// LS Electric XG5000 project: 과년67_2_4
// PLC NewPLC
// module base 0 slot 0: 입출력 모듈:XBC-DR20S (DC 24V 입력 12점, 릴레이 출력 8점)

PROGRAM NewProgram (task: 스캔 프로그램)

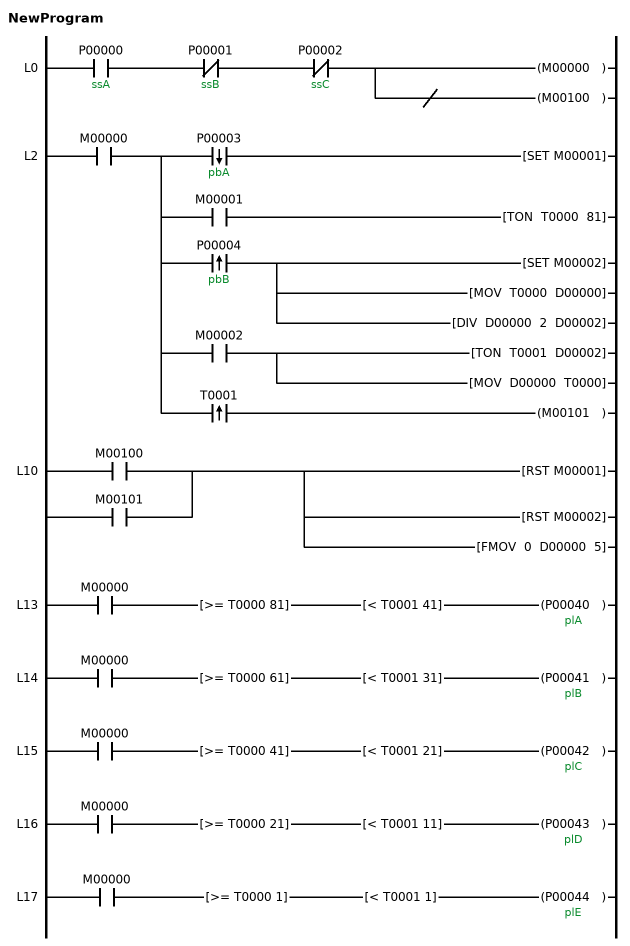
; L0
LOAD      P00000	// ssA
AND NOT   P00001	// ssB
AND NOT   P00002	// ssC
OUT       M00000
NOT
OUT       M00100
; L2
LOAD      M00000
MPUSH
ANDN      P00003	// pbA
SET       M00001
MLOAD
AND       M00001
TON       T0000 81
MLOAD
ANDP      P00004	// pbB
SET       M00002
MOV       T0000 D00000
DIV       D00000 2 D00002
MLOAD
AND       M00002
TON       T0001 D00002
MOV       D00000 T0000
MPOP
ANDP      T0001
OUT       M00101
; L10
LOAD      M00100
OR        M00101
RST       M00001
RST       M00002
FMOV      0 D00000 5
; L13
LOAD      M00000
AND>=     T0000 81
AND<      T0001 41
OUT       P00040	// plA
; L14
LOAD      M00000
AND>=     T0000 61
AND<      T0001 31
OUT       P00041	// plB
; L15
LOAD      M00000
AND>=     T0000 41
AND<      T0001 21
OUT       P00042	// plC
; L16
LOAD      M00000
AND>=     T0000 21
AND<      T0001 11
OUT       P00043	// plD
; L17
LOAD      M00000
AND>=     T0000 1
AND<      T0001 1
OUT       P00044	// plE

VARIABLES AND COMMENTS (devices not used above)
P00005	BIT	pbC